FUNCTION_BLOCK FB_CylinderTest EXTENDS FB_TestSuite
VAR
	fbCylinder : FB_Cylinder;
	
	masterMoveState, prevState : (
		init,
		runMoveToHomeTest,
		runPauseState,
		runMoveToWorkTest,
		cycleComplete,
		errorCycle
	);
	
	moveHomeTestState : (
		initToHome,
		requestCylinderMoveToHome,
		seeMovingToHomeStatus,
		waitForCylinderAtHome,
		completeToHome
	);
	moveToWorkTestState : (
		initToWork,
		requestCylinderMoveToWork,
		seeMovingToWorkStatus,
		waitForCylinderAtWork,
		completeToWork
	);
END_VAR

CycleCylinder();

METHOD CycleCylinder : int
VAR_INPUT
END_VAR
TEST('CycleCylinder');
CASE masterMoveState OF
	
	init:

		prevState := masterMoveState;
		masterMoveState := runMoveToHomeTest;
		
	runMoveToHomeTest :

		prevState := masterMoveState;
		IF MoveCylinderToHome() THEN
			masterMoveState := runPauseState;
		END_IF
		
	runPauseState:
		prevState := masterMoveState;
		masterMoveState := runMoveToWorkTest;
		
	runMoveToWorkTest :
	
		prevState := masterMoveState;
		IF MoveCylinderToWork() THEN
			masterMoveState := cycleComplete;
			
		END_IF
		
	cycleComplete :
		IF prevState <> masterMoveState THEN
			TEST_FINISHED_NAMED('CycleCylinder');
			prevState := masterMoveState;
		END_IF
		
END_CASE
END_METHOD

METHOD MoveCylinderToHome : BOOL
VAR_INST
	timeoutTimer : TON := (PT := fbCylinder.CYLINDER_MOVE_TIME + fbCylinder.CYLINDER_MOVE_TIME ); // allow twice the required time
END_VAR

CASE moveHomeTestState OF
	
	init:
		TEST('MoveCylinderToHome');
		moveHomeTestState := requestCylinderMoveToHome;
		
	requestCylinderMoveToHome :
		fbCylinder.MoveToHome();
		
		moveHomeTestState := seeMovingToHomeStatus;
		
	seeMovingToHomeStatus :
 
		AssertTrue( fbCylinder.MovingToHomePosition, 'fbCylinder.MovingToHome was not true');
		AssertTrue( fbCylinder.toHomePos, 'fbCylinder.toHomePos was not true');
		
		IF NOT ( fbCylinder.MovingToHomePosition AND fbCylinder.toHomePos ) THEN
			moveHomeTestState := waitForCylinderAtHome;
		ELSE
			moveHomeTestState := completeToHome;
		END_IF
		
	waitForCylinderAtHome :
	
		IF timeoutTimer.Q THEN
			moveHomeTestState := completeToHome;
			AssertTrue( FALSE , 'fbCylinder timed out moving to home.' );	
	
		ELSIF fbCylinder.AtHome THEN
			AssertTrue( TRUE , '' );
			moveHomeTestState := completeToHome;
			
			
		END_IF
		
	completeToHome :
		TEST_FINISHED_NAMED('MoveCylinderToHome');
		MoveCylinderToHome := TRUE;
END_CASE

timeoutTimer( IN := fbCylinder.MovingToHomePosition );
END_METHOD

METHOD MoveCylinderToWork : BOOL
VAR_INST
	timeoutTimer : TON := (PT := fbCylinder.CYLINDER_MOVE_TIME + fbCylinder.CYLINDER_MOVE_TIME ); // allow twice the required time
END_VAR

CASE moveToWorkTestState OF
	
	init:
		TEST('MoveCylinderToWork');
		moveToWorkTestState := requestCylinderMoveToWork;
		
	requestCylinderMoveToWork :
		fbCylinder.MoveToWork();
		
		moveToWorkTestState := seeMovingToWorkStatus;
		
	seeMovingToWorkStatus :
 
		AssertTrue( fbCylinder.MovingToWorkPosition, 'fbCylinder.MovingToWorkPosition was not true');
		AssertTrue( fbCylinder.toWorkPos, 'fbCylinder.toWorkPos was not true');
		
		IF NOT ( fbCylinder.MovingToHomePosition AND fbCylinder.toHomePos ) THEN
			moveToWorkTestState := waitForCylinderAtWork;
		ELSE
			moveToWorkTestState := completeToWork;
		END_IF
		
	waitForCylinderAtWork :
	
		IF timeoutTimer.Q THEN
			moveToWorkTestState := completeToWork;
			AssertTrue( FALSE , 'fbCylinder timed out moving to work.' );	
	
		ELSIF fbCylinder.AtWork THEN
			AssertTrue( TRUE , '' );
			moveToWorkTestState := completeToWork;
		
		END_IF
		
	completeToWork :
		TEST_FINISHED_NAMED('MoveCylinderToWork');
		MoveCylinderToWork := TRUE;
END_CASE

timeoutTimer( IN := fbCylinder.MovingToWorkPosition );
END_METHOD

END_FUNCTION_BLOCK

(* stored: Version 1.1.0.1, ProductVersion 3.1.4024.4
   POU FB_CylinderTest: Id {c9681de6-3801-4351-b3e3-1704c7faa79b}, SpecialFunc None
   Method CycleCylinder: Id {2f755462-1437-4939-92cb-0ec93d8f7e06}
   Method MoveCylinderToHome: Id {d1670a49-1575-44f3-8e2b-e20c2cb1c3ba}
   Method MoveCylinderToWork: Id {ac164537-900c-4f94-aea7-aab467983538} *)
